// TIA Portal project "BatteryStation" (V20)

(* hardware
DEVICE "S7-1500/ET200MP station_1"  S7-1500 station
   slot 0: "Rail_0"  Rack  6ES7 590-1***0-0AA0
   slot 1: "PLC_1"  CPU 1511-1 PN  6ES7 511-1AL03-0AB0  V3.1
      slot 3: "CPU display_1"  6ES7591-1AA00-0AA0
      slot 32768: "PROFINET interface_1"  X1
         slot 32769: "Port_1"  X1 P1
         slot 32770: "Port_2"  X1 P2
      slot 34817: "Virtual CP interface port_1"  Virtual CP interface port  Virtual CP interface port
DEVICE "HMI_1"  TP700 Comfort
   slot 0: "HMI_1"  TP700 Comfort  6AV2 124-0GC01-0AX0  17.0.0.0
   slot 1: "HMI_RT_1"  TP700 Comfort  6AV2 124-0GC01-0AX0  17.0.0.0
   slot 5: "HMI_1.IE_CP_1"  PROFINET Interface  17.0.0.0
      slot 1: "PROFINET Interface_1"  PROFINET Interface
         slot 1: "Port_1"  Port
         slot 2: "Port_2"  Port
   slot 7: "HMI_1.MPI/DP_CP_1"  MPI/DP Interface  17.0.0.0
*)

// ===== PLC "PLC_1"  CPU 1511-1 PN =====

VAR_GLOBAL   // PLC tag table "Default tag table"
   "PB_Start" AT %I0.0 : Bool;   // Start button
   "PB_Stop" AT %I0.1 : Bool;   // Stop button
   "PB_Reset" AT %I0.2 : Bool;   // Reset button
   "EStop_OK" AT %I0.3 : Bool;   // TRUE = E-stop NOT pressed
   "B1_ModuleAtStation" AT %I0.4 : Bool;   // Sensor: module at station
   "B2_ClampClosed" AT %I0.5 : Bool;   // Sensor: clamp closed
   "M1_Conveyor" AT %Q0.0 : Bool;   // Conveyor motor
   "Y1_Clamp" AT %Q0.1 : Bool;   // Clamp valve
   "H1_Running" AT %Q0.2 : Bool;   // Lamp: running
   "H2_Fault" AT %Q0.3 : Bool;   // Lamp: fault
   "H3_MaintenanceDue" AT %Q0.4 : Bool;   // Lamp: maintenance due
END_VAR

DATA_BLOCK "HMI"   // DB1
{ S7_Optimized_Access := 'TRUE' }
VERSION : 0.1
// ---------------------------------------------------------------------
//  DB "HMI": everything the operator screen reads and writes
//  ---------------------------------------------------------------------
   VAR
      StartBtn : Bool;   // HMI buttons (ON while pressed)
      StopBtn : Bool;
      ResetBtn : Bool;
      EStopBtn : Bool;   // simulated emergency stop (TRUE = pressed)
      ServiceDoneBtn : Bool;
      SimMode : Bool := TRUE;   // TRUE = use the fake machine
      SimJam : Bool;   // fault injection
      SimSensorFault : Bool;   // fault injection
      AlarmWord : Word;   // copied from the station for HMI alarms
   END_VAR
BEGIN
END_DATA_BLOCK

DATA_BLOCK "Station_DB"   // DB2
{ S7_Optimized_Access := 'TRUE' }
VERSION : 0.1
// stored: InstanceOfName FB_Station
"FB_Station"
BEGIN
END_DATA_BLOCK

DATA_BLOCK "PlantSim_DB"   // DB3
{ S7_Optimized_Access := 'TRUE' }
VERSION : 0.1
// stored: InstanceOfName FB_PlantSim
"FB_PlantSim"
BEGIN
END_DATA_BLOCK

FUNCTION_BLOCK "FB_Device"   // FB1, SCL
{ S7_Optimized_Access := 'TRUE' }
VERSION : 0.1
// =====================================================================
//  Battery Module Assembly Station - simulated maintenance demo
//  Siemens TIA Portal V20, S7-1500, SCL
//  Blocks: FB_Device (reusable, used twice), FB_PlantSim, FB_Station,
//          DB "HMI", instance DBs, FC_Main (called from OB1)
//  =====================================================================
//  ---------------------------------------------------------------------
//  FB_Device: ONE standard block for any device that is switched ON and
//  must confirm with a sensor (motor, valve, clamp...).
//  - switches the output only when allowed
//  - raises a FAULT if the sensor does not confirm in time (timeout)
//  - counts starts and running seconds (data for preventive maintenance)
//  ---------------------------------------------------------------------
   VAR_INPUT
      Cmd : Bool;   // sequence wants the device ON
      Feedback : Bool;   // sensor confirms the device did its job
      Timeout : Time := T#5S;   // max time allowed to get the feedback
      ResetCmd : Bool;   // operator reset of the fault
      Enable : Bool;   // FALSE = interlock (e.g. emergency stop)
   END_VAR
   VAR_OUTPUT
      Q : Bool;   // drive output (contactor / valve)
      Fault : Bool;   // timeout fault, stays ON until reset
   END_VAR
   VAR
      Operations : DInt;   // number of starts (maintenance data)
      OperatingTime_s : DInt;   // total ON time in seconds (maintenance data)
      tonTimeout : TON_TIME;
      tonSecond : TON_TIME;
      qOld : Bool;
   END_VAR
BEGIN

   // 1) Output ON only if commanded, enabled and not faulted
   #Q := #Cmd AND #Enable AND NOT #Fault;

   // 2) Count starts (rising edge of the output)
   IF #Q AND NOT #qOld THEN
       #Operations := #Operations + 1;
   END_IF;
   #qOld := #Q;

   // 3) Timeout supervision: ON but no feedback within Timeout -> fault
   #tonTimeout(IN := #Q AND NOT #Feedback,
               PT := #Timeout);
   IF #tonTimeout.Q THEN
       #Fault := TRUE;
   END_IF;

   // 4) Reset clears the fault
   IF #ResetCmd THEN
       #Fault := FALSE;
   END_IF;

   // 5) Running-time counter: +1 every second while ON
   #tonSecond(IN := #Q AND NOT #tonSecond.Q,
              PT := T#1S);
   IF #tonSecond.Q THEN
       #OperatingTime_s := #OperatingTime_s + 1;
   END_IF;
END_FUNCTION_BLOCK

FUNCTION_BLOCK "FB_PlantSim"   // FB2, SCL
{ S7_Optimized_Access := 'TRUE' }
VERSION : 0.1
// ---------------------------------------------------------------------
//  FB_PlantSim: a FAKE machine, so we can test without hardware.
//  It reacts to the PLC outputs and creates the sensor signals.
//  Two switches inject faults on purpose to test the alarms.
//  ---------------------------------------------------------------------
   VAR_INPUT
      ConveyorOn : Bool;
      ClampOn : Bool;
      SimJam : Bool;   // TRUE = module stuck, never arrives
      SimSensorFault : Bool;   // TRUE = clamp sensor broken
   END_VAR
   VAR_OUTPUT
      B1_ModuleAtStation : Bool;
      B2_ClampClosed : Bool;
   END_VAR
   VAR
      partAtStation : Bool;
      tonArrive : TON_TIME;
      tonLeave : TON_TIME;
      tonClamp : TON_TIME;
   END_VAR
BEGIN

   // Module travels 3 s on the conveyor until it reaches the station
   #tonArrive(IN := #ConveyorOn AND NOT #partAtStation AND NOT #SimJam,
              PT := T#3S);
   IF #tonArrive.Q THEN
       #partAtStation := TRUE;
   END_IF;

   // Module leaves the station 1.5 s after the conveyor restarts
   #tonLeave(IN := #ConveyorOn AND #partAtStation AND NOT #ClampOn,
             PT := T#1500MS);
   IF #tonLeave.Q THEN
       #partAtStation := FALSE;
   END_IF;

   // Clamp needs 0.8 s to close
   #tonClamp(IN := #ClampOn AND NOT #SimSensorFault,
             PT := T#800MS);

   #B1_ModuleAtStation := #partAtStation;
   #B2_ClampClosed := #tonClamp.Q;
END_FUNCTION_BLOCK

FUNCTION_BLOCK "FB_Station"   // FB3, SCL
{ S7_Optimized_Access := 'TRUE' }
VERSION : 0.1
// ---------------------------------------------------------------------
//  FB_Station: the station logic
//  Step 0 idle -> 10 transport in -> 20 clamp -> 30 process 2 s
//         -> 40 release + transport out -> back to 10
//  ---------------------------------------------------------------------
   VAR_INPUT
      StartCmd : Bool;
      StopCmd : Bool;
      ResetCmd : Bool;
      EStopOK : Bool;   // TRUE = emergency stop NOT pressed
      B1_ModuleAtStation : Bool;
      B2_ClampClosed : Bool;
      ServiceDone : Bool;   // technician confirms the service was done
   END_VAR
   VAR_OUTPUT
      M1_Conveyor : Bool;
      Y1_Clamp : Bool;
      H1_Running : Bool;
      H2_Fault : Bool;
      H3_MaintenanceDue : Bool;
      AlarmWord : Word;   // bit0 E-stop, bit1 conveyor timeout, bit2 clamp timeout, bit3 maintenance due
   END_VAR
   VAR
      "Step" : Int;   // current step of the sequence
      Running : Bool;
      EStopFault : Bool;
      Conveyor : "FB_Device";   // same standard block...
      Clamp : "FB_Device";   // ...used twice
      tonProcess : TON_TIME;
      tonCycle : TON_TIME;
      cycleDone : Bool;
      LastCycleTime : Time;
      CyclesTotal : DInt;
      CyclesSinceService : DInt;
      ServiceInterval : DInt := 20;   // demo value: service every 20 cycles
   END_VAR
   VAR_TEMP
      anyFault : Bool;
      convCmd : Bool;
      clampCmd : Bool;
   END_VAR
BEGIN

   // --- 1. Emergency stop: latched until Reset with the E-stop released
   IF NOT #EStopOK THEN
       #EStopFault := TRUE;
   ELSIF #ResetCmd THEN
       #EStopFault := FALSE;
   END_IF;

   #anyFault := #EStopFault OR #Conveyor.Fault OR #Clamp.Fault;

   // --- 2. Run latch (start/stop "seal-in"). Stop and faults win over Start.
   IF #StopCmd OR #anyFault THEN
       #Running := FALSE;
   ELSIF #StartCmd THEN
       #Running := TRUE;
   END_IF;

   IF NOT #Running THEN
       #Step := 0;
   END_IF;

   // --- 3. Sequence (step chain)
   #tonProcess(IN := (#Step = 30),
               PT := T#2S);
   #cycleDone := FALSE;

   CASE #Step OF
       0:  // Idle
           IF #Running THEN
               #Step := 10;
           END_IF;
       10: // Transport module in
           IF #B1_ModuleAtStation THEN
               #Step := 20;
           END_IF;
       20: // Close clamp
           IF #B2_ClampClosed THEN
               #Step := 30;
           END_IF;
       30: // Process (e.g. pressing / screwing) for 2 s
           IF #tonProcess.Q THEN
               #Step := 40;
           END_IF;
       40: // Open clamp, transport module out
           IF NOT #B1_ModuleAtStation AND NOT #B2_ClampClosed THEN
               #cycleDone := TRUE;
               #Step := 10;
           END_IF;
   END_CASE;

   // --- 4. Devices (same block, two instances)
   #convCmd := (#Step = 10) OR ((#Step = 40) AND NOT #B2_ClampClosed);
   #clampCmd := (#Step = 20) OR (#Step = 30);

   #Conveyor(Cmd := #convCmd,
             Feedback := ((#Step = 10) AND #B1_ModuleAtStation) OR ((#Step = 40) AND NOT #B1_ModuleAtStation),
             Timeout := T#8S,
             ResetCmd := #ResetCmd,
             Enable := NOT #EStopFault);

   #Clamp(Cmd := #clampCmd,
          Feedback := #B2_ClampClosed,
          Timeout := T#3S,
          ResetCmd := #ResetCmd,
          Enable := NOT #EStopFault);

   // --- 5. Cycle time and counters
   IF #cycleDone THEN
       #LastCycleTime := #tonCycle.ET;
       #CyclesTotal := #CyclesTotal + 1;
       #CyclesSinceService := #CyclesSinceService + 1;
   END_IF;
   #tonCycle(IN := (#Step <> 0) AND NOT #cycleDone,
             PT := T#1H);

   // --- 6. Preventive maintenance
   IF #ServiceDone THEN
       #CyclesSinceService := 0;
   END_IF;
   #H3_MaintenanceDue := #CyclesSinceService >= #ServiceInterval;

   // --- 7. Outputs and alarms
   #M1_Conveyor := #Conveyor.Q;
   #Y1_Clamp := #Clamp.Q;
   #H1_Running := #Running;
   #H2_Fault := #anyFault;

   #AlarmWord := W#16#0;
   #AlarmWord.%X0 := #EStopFault;
   #AlarmWord.%X1 := #Conveyor.Fault;
   #AlarmWord.%X2 := #Clamp.Fault;
   #AlarmWord.%X3 := #H3_MaintenanceDue;
END_FUNCTION_BLOCK

FUNCTION "FC_Main" : Void   // FC1, SCL
{ S7_Optimized_Access := 'TRUE' }
VERSION : 0.1
// ---------------------------------------------------------------------
//  FC_Main: wiring. Chooses real or simulated sensors, calls the blocks.
//  Called from OB1 (Main).
//  ---------------------------------------------------------------------
   VAR_TEMP
      b1 : Bool;
      b2 : Bool;
      estopOK : Bool;
   END_VAR
BEGIN

   // Sensors: from the fake machine (simulation) or from real inputs
   IF "HMI".SimMode THEN
       #b1 := "PlantSim_DB".B1_ModuleAtStation;
       #b2 := "PlantSim_DB".B2_ClampClosed;
       #estopOK := NOT "HMI".EStopBtn;
   ELSE
       #b1 := "B1_ModuleAtStation";
       #b2 := "B2_ClampClosed";
       #estopOK := "EStop_OK";
   END_IF;

   "Station_DB"(StartCmd := "PB_Start" OR "HMI".StartBtn,
                StopCmd := "PB_Stop" OR "HMI".StopBtn,
                ResetCmd := "PB_Reset" OR "HMI".ResetBtn,
                EStopOK := #estopOK,
                B1_ModuleAtStation := #b1,
                B2_ClampClosed := #b2,
                ServiceDone := "HMI".ServiceDoneBtn,
                M1_Conveyor => "M1_Conveyor",
                Y1_Clamp => "Y1_Clamp",
                H1_Running => "H1_Running",
                H2_Fault => "H2_Fault",
                H3_MaintenanceDue => "H3_MaintenanceDue",
                AlarmWord => "HMI".AlarmWord);

   "PlantSim_DB"(ConveyorOn := "M1_Conveyor",
                 ClampOn := "Y1_Clamp",
                 SimJam := "HMI".SimJam,
                 SimSensorFault := "HMI".SimSensorFault);
END_FUNCTION

ORGANIZATION_BLOCK "Main"   // OB1, LAD, ProgramCycle
TITLE = "Main Program Sweep (Cycle)"
{ S7_Optimized_Access := 'TRUE' }
VERSION : 0.1
   VAR_INPUT
      Initial_Call : Bool;   // Initial call of this OB
      Remanence : Bool;   // =True, if remanent data are available
   END_VAR
BEGIN

REGION Network 1
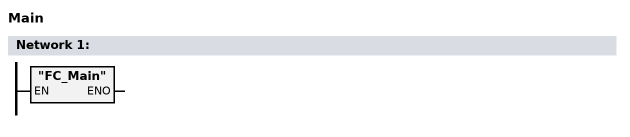
   RUNG wire#powerrail
      "FC_Main"()
   END_RUNG
   // the same network as SCL:
   "FC_Main"();
END_REGION
END_ORGANIZATION_BLOCK

(* ===== HMI "HMI_RT_1" =====
system functions are stored by id; their names below are inferred from use
connection "HMI_Connection_1": ETHERNET, S7_1500_OMS

HMI tags "Default tag table"
   "Tag_ScreenNumber" : UInt, internal
   "HMI_StartBtn" : Bool = PLC HMI.StartBtn, 1 s
   "HMI_StopBtn" : Bool = PLC HMI.StopBtn, 1 s
   "HMI_ResetBtn" : Bool = PLC HMI.ResetBtn, 1 s
   "HMI_ServiceDoneBtn" : Bool = PLC HMI.ServiceDoneBtn, 1 s
   "HMI_EStopBtn" : Bool = PLC HMI.EStopBtn, 1 s
   "HMI_SimJam" : Bool = PLC HMI.SimJam, 1 s
   "HMI_SimSensorFault" : Bool = PLC HMI.SimSensorFault, 1 s
   "H1_Running" : Bool = PLC H1_Running AT %Q0.2, 1 s
   "H2_Fault" : Bool = PLC H2_Fault AT %Q0.3, 1 s
   "H3_MaintenanceDue" : Bool = PLC H3_MaintenanceDue AT %Q0.4, 1 s
   "Station_DB_Step" : Int = PLC Station_DB.Step, 1 s
   "Station_DB_CyclesSinceService" : DInt = PLC Station_DB.CyclesSinceService, 1 s
   "Station_DB_LastCycleTime" : Time = PLC Station_DB.LastCycleTime, 1 s
   "Station_DB_AlarmWord" : Word = PLC Station_DB.AlarmWord, 1 s

discrete alarms
   1: 'EMERGENCY STOP pressed', class Errors, trigger "Station_DB_AlarmWord" bit 0
   2: 'CONVEYOR JAM - module not arrived', class Errors, trigger "Station_DB_AlarmWord" bit 1
   3: 'CLAMP SENSOR FAULT - no feedback', class Errors, trigger "Station_DB_AlarmWord" bit 2
   4: 'MAINTENANCE DUE - service the station', class Warnings, trigger "Station_DB_AlarmWord" bit 3

screen "Root screen" 800x420, template "Template_1"
   on GenerateScreen: SetTag("Tag_ScreenNumber", 1)
   Button "Button_1" at 15,85 size 130x50; TextOff 'START'
      on Press: SetBit("HMI_StartBtn")
      on Release: ResetBit("HMI_StartBtn")
   Button "Button_2" at 15,145 size 130x50; TextOff 'STOP'
      on Press: SetBit("HMI_StopBtn")
      on Release: ResetBit("HMI_StopBtn")
   Button "Button_3" at 15,205 size 130x50; TextOff 'RESET'
      on Press: SetBit("HMI_ResetBtn")
      on Release: ResetBit("HMI_ResetBtn")
   Button "Button_4" at 15,345 size 130x50; TextOff 'SERVICE DONE'
      on Press: SetBit("HMI_ServiceDoneBtn")
      on Release: ResetBit("HMI_ServiceDoneBtn")
   Button "Button_5" at 15,265 size 130x50; TextOff 'E-STOP'
      on Click: InvertBit("HMI_EStopBtn")
   Button "Button_6" at 165,345 size 125x50; TextOff 'SIM: JAM'
      on Click: InvertBit("HMI_SimJam")
   Button "Button_7" at 300,345 size 125x50; TextOff 'SIM: SENSOR'
      on Click: InvertBit("HMI_SimSensorFault")
   Circle "Circle_1" at 170,90 size 32x32
      Appearance <- "H1_Running"
   Circle "Circle_2" at 170,135 size 32x32
      Appearance <- "H2_Fault"
   Circle "Circle_3" at 170,180 size 32x32
      Appearance <- "H3_MaintenanceDue"
   TextField "Text field_1" at 210,97 size 91x23; Text 'RUNNING'
   TextField "Text field_2" at 210,142 size 63x23; Text 'FAULT'
   TextField "Text field_3" at 210,187 size 182x23; Text 'MAINTENANCE DUE'
   TextField "Text field_4" at 170,237 size 53x23; Text 'Step:'
   TextField "Text field_5" at 170,272 size 191x23; Text 'Cycles since service:'
   TextField "Text field_6" at 170,307 size 148x23; Text 'Last cycle [ms]:'
   TextField "Text field_7" at 15,55 size 360x23; Text 'BATTERY MODULE ASSEMBLY STATION'
   IOField "I/O field_1" at 350,230 size 90x28; FormatPattern s99999
      ProcessValue <- "Station_DB_Step"
   IOField "I/O field_2" at 350,265 size 90x28; FormatPattern s9999999999
      ProcessValue <- "Station_DB_CyclesSinceService"
   IOField "I/O field_3" at 350,300 size 90x28; FormatPattern s9999999999
      ProcessValue <- "Station_DB_LastCycleTime"
   AlarmView "Alarm view_1" at 445,85 size 345x330

Template "Template_1" 800x420
   Button "Exit" at 720,360 size 78x58; TextOff 'Exit'; PictureOff "ExitRuntime_TP700_Comfort_TR"; PictureOn "ExitRuntime_TP700_Comfort_TR"
      on Release: StopRuntime(0)
   Button "Template_Button" at 640,360 size 78x58; TextOff 'Text'
   Button "Template_Button_1" at 560,360 size 78x58; TextOff 'Text'
   Button "Template_Button_2" at 480,360 size 78x58; TextOff 'Text'
   Button "Template_Button_3" at 400,360 size 78x58; TextOff 'Text'
   Button "Template_Button_4" at 321,360 size 78x58; TextOff 'Text'
   Button "Template_Button_5" at 241,360 size 78x58; TextOff 'Text'
   Button "Template_Button_6" at 161,360 size 78x58; TextOff 'Text'
   Button "Template_Button_7" at 81,360 size 78x58; TextOff 'Text'
   Button "Start screen" at 1,360 size 78x58; TextOff 'Start screen'; PictureOff "NavigateHome_TP700_Comfort_TR"; PictureOn "NavigateHome_TP700_Comfort_TR"
      on Release: ActivateScreen("Root screen", 0)
*)